PROGRAM MAIN
VAR
	bInit		: BOOL;
	arrData		: ARRAY[0..2] OF UINT;
	
	
	
	
	
	
	
	
	
	
	
	
END_VAR

END_PROGRAM

(* stored: Version 1.1.0.1, ProductVersion 3.1.4024.15
   POU MAIN: Id {768887be-c808-4342-97c7-6a09e98fd057}, SpecialFunc None *)
